// Queue-based Modbus RTU command handler with ringbuffer
{attribute 'no_explicit_call' := 'do not call this POU directly'}
FUNCTION_BLOCK ModbusHandler_KL6x22B IMPLEMENTS I_ModbusHandler
VAR_INPUT
END_VAR
VAR_OUTPUT
END_VAR
VAR
	_Terminal							: Tc2_ModbusRTU.ModbusRtuMasterV2_KL6x22B;
END_VAR
VAR
	_Busy								: BOOL;
	_Error								: BOOL;
	_ErrorId								: MODBUS_ERRORS;
	_ModbusTimeout						: TIME := T#500MS;	
	_commandToProcess					: ST_ModbusCommand;
	_bufferHandler						: Tc3_AnyBuffer.FifoBuffer(_buffer,TRUE,FALSE);
	_buffer								: Tc3_AnyBuffer.AnyBuffer(_arBuffer,0,param.MAXMODBUSBUFFER,FALSE);
	_arBuffer							: ARRAY[0..MAXMODBUSBUFFER] OF ST_ModbusCommand;
	_bufferLock							: BOOL;
END_VAR
VAR CONSTANT
	ERROR_RESULT						: hresult := e_fail;
	OK_RESULT							: hresult := s_ok;
END_VAR

METHOD AddToBuffer : Hresult
VAR_INPUT
	command			: ST_ModbusCommand;
END_VAR
VAR CONSTANT
	PENDING_RESULT		: hresult := S_Pending;
END_VAR
// Set status to pending and add to ringbuffer
IF Tc2_System.TestAndSet(_bufferLock) THEN
	MEMCPY(destAddr:= command.Result,srcAddr:=ADR(PENDING_RESULT),n:=SIZEOF(PENDING_RESULT));
	_bufferHandler.Push(command);
	
	AddToBuffer := s_ok;
	_bufferLock:=FALSE;
ELSE
	AddToBuffer := e_fail;
END_IF
END_METHOD

PROPERTY Busy : bool
GET
Busy			:= _Busy;
END_GET
END_PROPERTY

METHOD Cyclic
(*----------------------------------------------------------------------
Wait for a new bufferd command to process
-----------------------------------------------------------------------*)
	// Check for queued commands
	IF NOT _Busy AND NOT _bufferLock THEN
		IF NOT _bufferHandler.isEmpty THEN
			_Error := FALSE;
			_ErrorId	:= 0;
			_Busy								:= _bufferHandler.Pop(_commandToProcess);
		END_IF
	END_IF
		
	(*----------------------------------------------------------------------
	Process command
	-----------------------------------------------------------------------*)
	IF _Busy AND _commandToProcess.Result <> 0 THEN
			// Copy parameters to modbus FB
			_Terminal.UnitID    		:= _commandToProcess.UnitID;
			_Terminal.Quantity  		:= _commandToProcess.Quantity;
			_Terminal.MBAddr    		:= _commandToProcess.MBAddr;
			_Terminal.cbLength		:= _commandToProcess.cbLength;
			_Terminal.Timeout			:= _ModbusTimeout;
			_Terminal.pMemoryAddr 	:= _commandToProcess.pMemoryAddr;

		CASE _commandToProcess.ModbusFunction OF
			E_ModbusFunction.ReadCoils:
				_Terminal.readcoils(	execute := TRUE,
									);
			E_ModbusFunction.ReadInputStatus:
				_Terminal.ReadInputStatus(execute := TRUE,
									);
			E_ModbusFunction.ReadRegs	:
				_Terminal.ReadRegs(execute := TRUE,
									);
			E_ModbusFunction.ReadInputRegs :
				_Terminal.ReadInputRegs(execute := TRUE,
									);
			E_ModbusFunction.WriteSingleCoil:
				_Terminal.WriteSingleCoil(execute := TRUE);
			E_ModbusFunction.WriteSingleRegister:
				_Terminal.WriteSingleRegister(execute := TRUE);
			E_ModbusFunction.WriteMultipleCoils	:
				_Terminal.WriteMultipleCoils(execute := TRUE);
			E_ModbusFunction.WriteRegs		:
				_Terminal.WriteRegs(execute := TRUE);
			E_ModbusFunction.Diagnostics		:
				_Terminal.Diagnostics(execute := TRUE);

		END_CASE
			// Wait for completion
			IF NOT _Terminal.BUSY THEN
				
				_Terminal.readcoils(	execute := FALSE,);
				_Terminal.ReadInputStatus(execute := FALSE,);
				_Terminal.ReadRegs(execute := FALSE,);
				_Terminal.ReadInputRegs(execute := FALSE,);
				_Terminal.WriteSingleCoil(execute := FALSE);
				_Terminal.WriteSingleRegister(execute := FALSE);
				_Terminal.WriteMultipleCoils(execute := FALSE);
				_Terminal.WriteRegs(execute := FALSE
				_Terminal.Diagnostics(execute := false);
				
				_Busy									:= FALSE;
				// Write result to caller's pointer
				IF NOT _Terminal.Error THEN
					MEMCPY(destAddr:= _commandToProcess.Result,srcAddr:=ADR(OK_RESULT),n:=SIZEOF(OK_RESULT));
				ELSE
					MEMCPY(destAddr:= _commandToProcess.Result,srcAddr:=ADR(ERROR_RESULT),n:=SIZEOF(ERROR_RESULT));
					//ADSLOGSTR( msgCtrlMask := ADSLOG_MSGTYPE_ERROR, msgFmtStr := 'modbus command Failed', strArg :='');
					_Error := TRUE;
					_ErrorId	:= _Terminal.ErrorId;
				END_IF
			END_IF
		ELSIF _Busy AND _commandToProcess.Result <> 0 THEN
			//ADSLOGSTR( msgCtrlMask := ADSLOG_MSGTYPE_ERROR, msgFmtStr := 'bad command receieved', strArg :='');
			_Busy		:= FALSE;
		END_IF
END_METHOD

PROPERTY Error : bool
GET
Error		:= _Error;
END_GET
END_PROPERTY

PROPERTY Errorid : MODBUS_ERRORS
GET
Errorid		:= _ErrorId;
END_GET
END_PROPERTY

PROPERTY ModbusTimeout : Time
SET
_ModbusTimeout		:=ModbusTimeout;
END_SET
END_PROPERTY

END_FUNCTION_BLOCK

(* stored: Version 1.1.0.1
   POU ModbusHandler_KL6x22B: Id {813ed012-1448-4a77-9239-d5e09ab2f179}, SpecialFunc None
   Method AddToBuffer: Id {28c798d7-9f5a-40f1-868f-4a6e50174de6}
   Property Busy: Id {a7a1f103-d7b6-44d4-9f7e-ddd7859f15c2}
   Get Get: Id {883cc578-a3d0-45f8-acbf-ca3dea5160d4}
   Method Cyclic: Id {1c26d61e-e260-4216-8442-265b33cb0637}
   Property Error: Id {d5b1f9f8-2939-491b-a182-00c607bac874}
   Get Get: Id {a8ada186-03ff-460e-bffc-6872d9e3e7f4}
   Property Errorid: Id {fa2689e9-0962-4924-bce9-4b64b7bc7604}
   Get Get: Id {75bbc25c-52d2-4f34-9a39-1c8944fe6048}
   Property ModbusTimeout: Id {d16fef32-8dd0-4055-9d24-023356519ad3}
   Set Set: Id {12f8d00c-1e87-4fe6-9d1b-0595d67842ee} *)
